FUNCTION_BLOCK I_COGSOGRapidUpdate (* This parameter group is a single frame parameter group that provides Course Over Ground (COG) and Speed Over Ground (SOG) *)
  (* Standard: NMEA 2000; Classification: PGN 129026; Function: COG & SOG, Rapid Update; Description: Copyright (c) 2024 HR Agrartechnik GmbH This program and the accompanying materials are made available under the terms of the Eclipse Public License 2.0 which is available at https://www.eclipse.org/legal/epl-2.0/ SPDX-License-Identifier: EPL-2.0 *)
  (* Version 1.0, 07.02.2025, Moritz Ortmeier, HR Agrartechnik GmbH *)
  PACKAGE isobus::tecu;
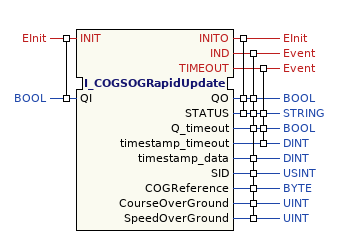
  EVENT_INPUT
    INIT : EInit WITH QI; (* Service Initialization *)
  END_EVENT
  EVENT_OUTPUT
    INITO : EInit WITH QO, STATUS; (* Initialization Confirm *)
    IND WITH QO, timestamp_data, SID, COGReference, STATUS, Q_timeout, CourseOverGround, SpeedOverGround; (* Indication from Resource *)
    TIMEOUT WITH timestamp_timeout, STATUS, Q_timeout;
  END_EVENT
  VAR_INPUT
    QI : BOOL; (* Event Input Qualifier *)
  END_VAR
  VAR_OUTPUT
    QO : BOOL; (* Event Output Qualifier *)
    STATUS : STRING;
    Q_timeout : BOOL;
    timestamp_timeout : DINT;
    timestamp_data : DINT;
    SID : USINT := USINT#16#FF; (* Sequence ID identifies the sequence this data is associated with so that the data can be synchronized with other vessel data for this same sequence being sent in another PGN. *)
    COGReference : BYTE := BYTE#16#FF; (* COG Reference--this field is used to indicate the direction reference of the course over ground. True North reference = 0. *)
    CourseOverGround : UINT := UINT#16#FFFF; (* Course Over Ground--this field is used to indicate the course over ground (COG) in resolution of 1x10-4 radians. *)
    SpeedOverGround : UINT := UINT#16#FFFF; (* Speed Over Ground--this field is used to indicate the speed over ground (SOG) in resolution of 1x10-2 meters/second. *)
  END_VAR
END_FUNCTION_BLOCK
